FUNCTION TryConvert_BYTE_TO_REAL : BOOL
VAR_INPUT
	in : BYTE;
	out : REFERENCE TO REAL;
END_VAR

out := BYTE_TO_REAL(in);
TryConvert_BYTE_TO_REAL := TRUE;

END_FUNCTION

(* stored: Version 1.1.0.1, ProductVersion 3.1.4024.12
   POU TryConvert_BYTE_TO_REAL: Id {44b4c8dd-602f-4ea1-9654-94f3258c1279}, SpecialFunc None *)
